// TIA Portal V21 export
DATA_BLOCK "DB611"   // DB611
TITLE = DB611
AUTHOR : PRECISE
FAMILY : PRECISE
// CIP AIR PURGING
// stored: AutoNumber false, InstanceOfName FB611, InstanceOfType FB
"FB611"
   // VAR_INPUT
   //    CycleEnable : Bool;
   //    CycleRunning : Bool;
   //    SecPulse : Bool;
   //    AlwaysTrue : Bool;
   //    ActualTemperature : Real;
   //    ActualPressure : Real;
   //    ActualRepetition : Int;
   //    ParaIn : "AirPurgingInputs";
   // END_VAR
   // VAR_OUTPUT
   //    Started : Bool;
   //    UtilityValve : Bool;
   //    VentValve : Bool;
   //    ParaOut : "AirPurgingOutputs";
   //    StepStatus : String[60];
   //    TempValve : Bool;
   //    TempValve_close : Bool;
   // END_VAR
   // VAR_IN_OUT
   //    Over : Bool;
   //    OverTemp : Bool;
   //    PressurePostiveTol : Real;
   //    PressureNegativeTol : Real;
   //    ControlStarted : Bool;
   //    TempPostiveTol : Real;
   //    TempNegativeTol : Real;
   //    HotAirValve : Bool;
   //    PopupSel : Bool;
   //    Popup : Bool;
   //    PopupAck : Bool;
   //    ControlStartedTemp : Bool;
   //    re_5 : Bool;
   //    TempReached : Bool;
   //    re_6 : Bool;
   // END_VAR
   // VAR
   //    ValveOnDelayPV : Int;
   //    ValveOffDelayPV : Int;
   //    RE1 : Bool;
   //    StepDelay { S7_SetPoint := 'True'} : "FB110";
   //    VentTimer { S7_SetPoint := 'True'} : "FB101";
   // END_VAR
BEGIN
   ParaIn.Selections.PressureMode := 1;
END_DATA_BLOCK
